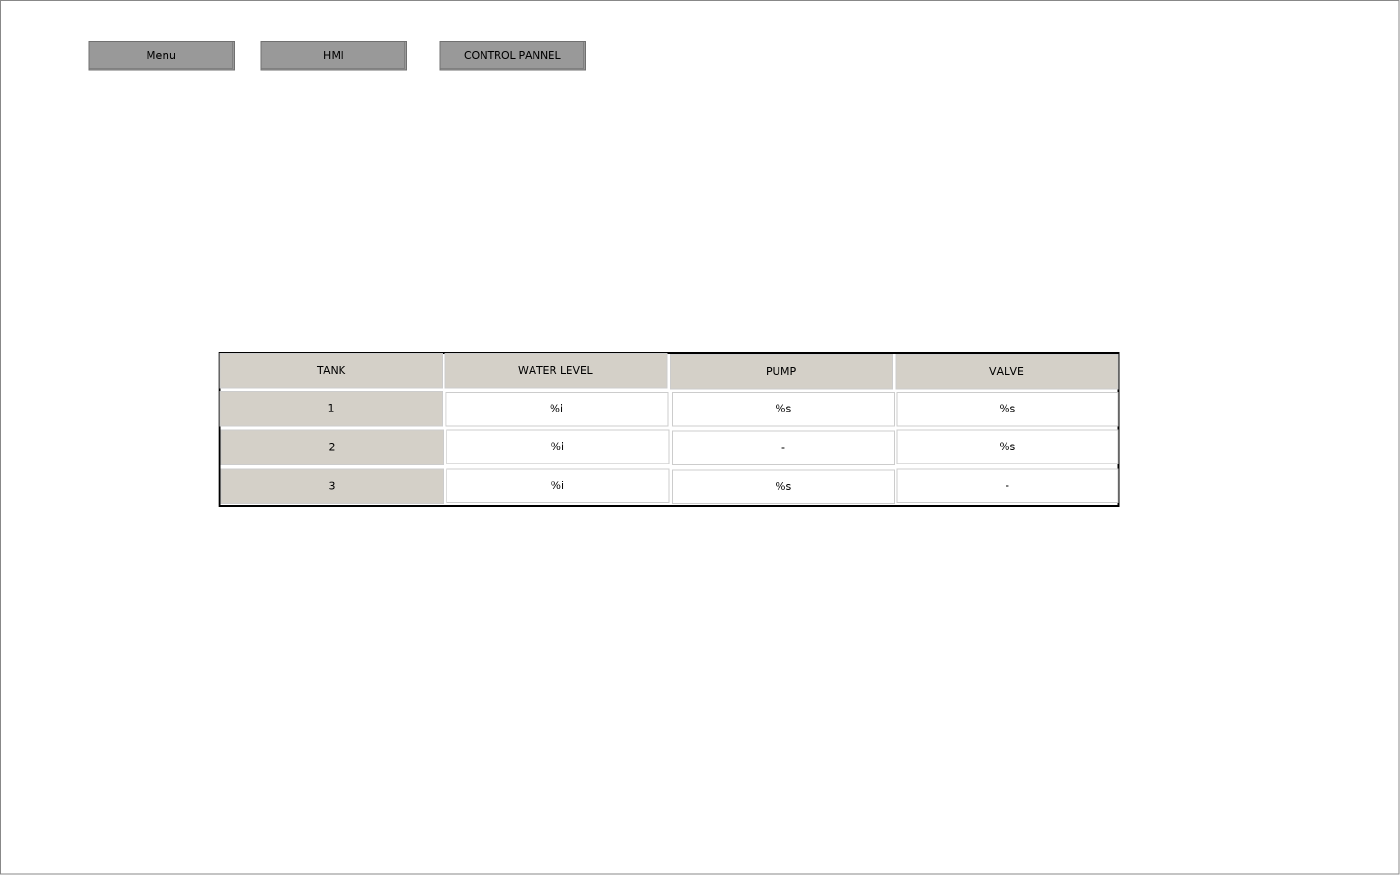
VISUALIZATION Pannello_Controllo  // 1440x900
    Button (91,42 150x30), "Menu"
        OnMouseClick: change screen: Menu
    Button (268,42 150x30), "HMI"
        OnMouseClick: change screen: Visualization
    Button (452,42 150x30), "CONTROL PANNEL"
        OnMouseClick: change screen: Pannello_Controllo
    Rectangle (225,362 926x159)
    Textfield (458,403 229x35), "%i", text variable: HMI.level_1
    Textfield (226,363 229x36), "TANK"
    Textfield (457,363 229x36), "WATER LEVEL"
    Textfield (689,364 229x36), "PUMP"
    Textfield (921,364 229x36), "VALVE"
    Textfield (226,402 229x36), "1"
    Textfield (227,442 229x36), "2"
    Textfield (227,482 229x36), "3"
    Textfield (459,442 229x35), "%i", text variable: HMI.level_2
    Textfield (459,482 229x35), "%i", text variable: HMI.level_3
    Textfield (691,403 229x35), "%s", text variable: HMI.pump_1
    Textfield (691,443 229x35), "-"
    Textfield (691,483 229x35), "%s", text variable: HMI.pump_3
    Textfield (922,403 228x35), "%s", text variable: HMI.valve
    Textfield (922,442 228x35), "%s", text variable: HMI.valve
    Textfield (922,482 228x35), "-"
END_VISUALIZATION

(* stored: Version 1.1.0.1
   Visu Pannello_Controllo: Id {4744b783-93a3-48bc-93ea-5332a9c2933b} *)
